(* IEC 61131-3 sources: Structured-Text/Source Code/Logic/LTA, 2 files *)

(* ---- Local Variables.ST ---- *)
VAR_INPUT
	IN_1:	REAL;		//Input Value
	IN_2:	REAL;		//Value the input will be compared against
	DEADBAND:	REAL;	//Size of the Deadband in units
END_VAR

VAR_OUTPUT
	OUT:	BOOL;
END_VAR

(* ---- LTA.ST ---- *)
//Mimics the logic of Honeywell CEE 'LT' less than block.

//Check if IN_1 is greater than IN_2.
IF IN_1 < IN_2 THEN
	OUT := TRUE;
END_IF;

//Reset OUT if it was previously TRUE and if IN_1 is less than IN_2 minus the deadband.
IF OUT AND IN_1 > (IN_2 + DEADBAND) THEN
	OUT := FALSE;
END_IF;
